{attribute 'qualified_only'}
{attribute 'strict'}
TYPE ePowerModuleThrottlingState :
(
	None := 0,
	FilterTemp := 1,
	InverterTemp:= 2,
	Overvoltage := 3
);
END_TYPE

(* stored: Version 1.1.0.1, ProductVersion 3.1.4026.18
   DUT ePowerModuleThrottlingState: Id {dcccd83d-1c30-4525-9324-91a9ce1b46d2} *)
